{attribute 'GeneratedUsingTerminal: EPP1332-0001-0016'}
{attribute addProperty BoxType "EPP1332-0001-0016"}
{attribute addProperty Id "EtcSlaveTerminalBaseInfoDataAT %I*InfoData_6F19DB2B2"}
{attribute addProperty CRC "2874840167"}
{attribute addProperty Size "2"}
TYPE EPP1332_AB5A9467 EXTENDS EtcSlaveTerminalBase :
STRUCT
	{attribute addProperty Name "InfoData"}
	InfoData : InfoData_6F19DB2B;
END_STRUCT
END_TYPE

(* stored: Version 1.2.0.0, ProductVersion 3.1.4024.9
   DUT EPP1332_AB5A9467: Id {de106db9-c09b-4476-852c-c83bd2a01163} *)
